Staubli VAL3: onStart.pgx

public program onStart(string& x_sItem[] (dimensions=1))
  local string l_sType
  local num i
  local string l_sPath
  local num l_nResult
  local string l_sName
begin

end
